Fanuc KAREL source: kb00110.KL

-- PROVISIONAL review KL for V1013-1; original PC SHA256 a4484854dba363531c7a94954790276ab8bf6310127d74a8bf72956b158b2781
-- Incomplete behavior may be omitted. Consult companion uncertainty JSON. Do not deploy.
PROGRAM KB00110
%NOLOCKGROUP
BEGIN
  -- UNRESOLVED_PC offsets 5-12; opcodes 9D,23
  -- UNRESOLVED_PC offsets 17-24; opcodes 9D,23
  -- UNRESOLVED_PC offsets 29-36; opcodes 9D,23
  -- UNRESOLVED_PC offsets 41-48; opcodes 9D,23
  -- UNRESOLVED_PC offsets 53-81; opcodes 27,22,22,22,22,31
  -- UNRESOLVED_PC offsets 86-90; opcodes 7F
END KB00110
